{attribute 'linkalways'} 
{attribute 'no_explicit_call' := 'This FB is a CLASS and must be accessed using methods or properties'}
{attribute 'enable_dynamic_creation'}
FUNCTION_BLOCK _GVCP_REGISTER_ADDRESS EXTENDS AliasDatatypeBase
VAR
	localData : GVCP_REGISTER_ADDRESS;
	activeData : REFERENCE TO GVCP_REGISTER_ADDRESS REF= localData;
	aliasBaseDatatype : _UDINT(0);
END_VAR

PROPERTY PUBLIC Address : PVOID
GET
Address := ADR(activeData);
END_GET
END_PROPERTY

METHOD PUBLIC ClearReference
VAR_INPUT
END_VAR
activeData REF= localData;
SetBaseDatatypeReference();
END_METHOD

METHOD PUBLIC Clone : I_Datatype
VAR
    pClone : POINTER TO _GVCP_REGISTER_ADDRESS;
END_VAR
pClone := __NEW(_GVCP_REGISTER_ADDRESS(InitialValue := Value));
Clone := pClone^;
END_METHOD

METHOD FB_init : BOOL
VAR_INPUT
	bInitRetains : BOOL; // if TRUE, the retain variables are initialized (warm start / cold start)
	bInCopyCode : BOOL;  // if TRUE, the instance afterwards gets moved into the copy code (online change)
	InitialValue : GVCP_REGISTER_ADDRESS; // if possible, not all values can be initialized
END_VAR
localData := InitialValue;
SetBaseDatatypeReference();
AddBaseDatatype(aliasBaseDatatype);
END_METHOD

PROPERTY PUBLIC Identifier : T_MAXSTRING
GET
Identifier := 'GVCP_REGISTER_ADDRESS';
END_GET
END_PROPERTY

METHOD PUBLIC MakeReferenceTo
VAR_INPUT
	ReferenceTarget : REFERENCE TO GVCP_REGISTER_ADDRESS;
END_VAR
activeData REF= ReferenceTarget;
SetBaseDatatypeReference();
END_METHOD

METHOD PROTECTED SetBaseDatatypeReference
VAR_INPUT
END_VAR
aliasBaseDatatype.MakeReferenceTo(activeData);
END_METHOD

PROPERTY PUBLIC Size : UDINT
GET
Size := SIZEOF(activeData);
END_GET
END_PROPERTY

METHOD TryMakeReferenceTo : BOOL
VAR_INPUT
	Target : I_Datatype;
END_VAR
VAR
	pTargetData : POINTER TO GVCP_REGISTER_ADDRESS;
END_VAR
IF NOT IsEquivalentTo(Target) THEN
	RETURN;
END_IF

pTargetData := Target.Address;
activeData REF= pTargetData^;
SetBaseDatatypeReference();
TryMakeReferenceTo := TRUE;
END_METHOD

PROPERTY PUBLIC Value : REFERENCE TO GVCP_REGISTER_ADDRESS
GET
Value REF= activeData;
END_GET
END_PROPERTY

END_FUNCTION_BLOCK

(* stored: Version 1.1.0.1, ProductVersion 3.1.4026.19
   POU _GVCP_REGISTER_ADDRESS: Id {0c77f638-088a-0cbe-0d83-00210d1ca2b2}, SpecialFunc None
   Folder Core: Id {d0955c98-6e25-0612-1130-c9f140b30a8b}
   Folder Protected: Id {b8aeb66d-5dc6-0e2c-270e-b562e5c9f5b5}
   Folder Customize: Id {b89f2593-6879-0cd8-2a33-c0acae44025a}
   Folder Constructor: Id {9e7e0138-649b-07d7-3c58-3b69b38c98fc}
   Property Address: Id {ba85c286-d2c4-01ec-3a39-23358f2d902a}
   Get Get: Id {7dd36d41-25a2-0a4c-021e-13c0abfd16c7}
   Method ClearReference: Id {64f78287-cd8f-0cdc-13e0-eedcf20fc197}
   Method Clone: Id {313db5dc-c1c6-0c3c-3021-ed2084bca227}
   Method FB_init: Id {547d8dfb-522d-03fe-0039-be25aabea986}
   Property Identifier: Id {975e137e-f986-0d9f-39d6-7a2663472d62}
   Get Get: Id {b5ac52b0-8aa3-08a8-0d24-e377bcc78596}
   Method MakeReferenceTo: Id {c1f8b00a-062e-0415-3290-0e730baf35e0}
   Method SetBaseDatatypeReference: Id {b921d901-3a13-0ce3-0790-d3457ac5b3fd}
   Property Size: Id {e587f4b1-5c1f-09e5-1d3b-1e58c0a581b2}
   Get Get: Id {5a0159f8-dfdd-02d2-11de-6617b7d8ca68}
   Method TryMakeReferenceTo: Id {ac52910f-f7fa-077c-3e4c-d1b6d4ef2047}
   Property Value: Id {6aaeccbf-4d5d-033d-239a-7cd66873059a}
   Get Get: Id {d1870a56-92df-034d-30ba-3257dae16b2e} *)
